// SIMATIC S7-200 project (STEP 7-Micro/WIN), CPU 224 REL 02.01

ORGANIZATION_BLOCK MAIN:OB1
TITLE=PROGRAM COMMENTS
BEGIN
Network 1 // Network Title
// VW0 - roznica temp
LD     I0.0
MOVW   +250, VW0
-I     AIW8, VW0
Network 2
// VW2 -> -k
// (network saved uncompiled; FBD cells follow)
// row 0: c1 [SUB_I ]
// row 1: c1 [ EN:=I0.0, IN1:=0, IN2:=+2, ENO=>V?0, OUT=>VW2]
// row 2: c1 [box]
// row 3: c1 [box]
Network 3
// VW4 - MOC WENT
LD     I0.0
MOVW   VW0, VW4
*I     VW2, VW4
Network 4
// WLACZ WENT
// (network saved uncompiled; FBD cells follow)
// row 0: c3 [MOV_W ]
// row 1: c1 [>I VW4 0 ]  c2 --  c3 [ EN:=power@row1, IN:=VW4, ENO=>V?0, OUT=>AQW0]
// row 2: c1 [box]  c3 [box]
Network 5
// WYLACZ WENT
// (network saved uncompiled; FBD cells follow)
// row 0: c3 [MOV_W ]
// row 1: c1 [>=I 0 VW4 ]  c2 --  c3 [ EN:=power@row1, IN:=0, ENO=>V?0, OUT=>AQW0]
// row 2: c1 [box]  c3 [box]
Network 6
// V1.0 - STAN ZAROWKI
LDW>   VW0, 0
=      V1.0
Network 8
// WLACZ ZAROWKE
// (network saved uncompiled; FBD cells follow)
// row 0: c3 [SUB_I ]
// row 1: c1 [AND I0.0 V1.0 ]  c2 --  c3 [ EN:=power@row1, IN1:=0, IN2:=1, ENO=>V?0, OUT=>VW4]
// row 2: c1 [box]  c3 [box]
// row 3: c3 [box]
Network 9
// WYLACZ ZAROWKE
// (network saved uncompiled; FBD cells follow)
// row 0: c3 [SUB_I ]
// row 1: c1 [AND I0.0 V1.0 ]  c2 --  c3 [ EN:=power@row1, IN1:=1, IN2:=0, ENO=>V?0, OUT=>VW4]
// row 2: c1 [box]  c3 [box]
// row 3: c3 [box]
Network 10
LDW<   VW4, 0
=      Q0.2
END_ORGANIZATION_BLOCK
